FUNCTION_BLOCK FB_ObjectExt EXTENDS FB_Object IMPLEMENTS ITF_ObjectExt
VAR_INPUT
END_VAR
VAR_OUTPUT
END_VAR
VAR
END_VAR

METHOD AddSomeValues : int
VAR_INPUT
	x : INT;
	y : INT;
END_VAR
AddSomeValues := x + y;
END_METHOD

END_FUNCTION_BLOCK

(* stored: Version 1.1.0.1, ProductVersion 3.1.4024.11
   POU FB_ObjectExt: Id {f6144f08-4245-4a22-86cd-bc3bb32680cc}, SpecialFunc None
   Method AddSomeValues: Id {8e26ebe2-fffe-429f-baa7-d1cca7448623} *)
